% RSLogix 500 project TRAFFIC Multiple.RSS, saved by version 8.30.00.16 %
PROJECT "UNTITLED"    % processor: Bul.1763 MicroLogix 1100 Series B %

PROGRAM FILES
  LAD 2   8 rungs

DATA FILES
  O0 OUTPUT  4 elements
  I1 INPUT  6 elements
  S2 STATUS  66 elements
  B3 BINARY  1 elements
  T4 TIMER  7 elements
  C5 COUNTER  1 elements
  R6 CONTROL  1 elements
  N7 INTEGER  1 elements
  F8 FLOAT  1 elements

LADDER 2
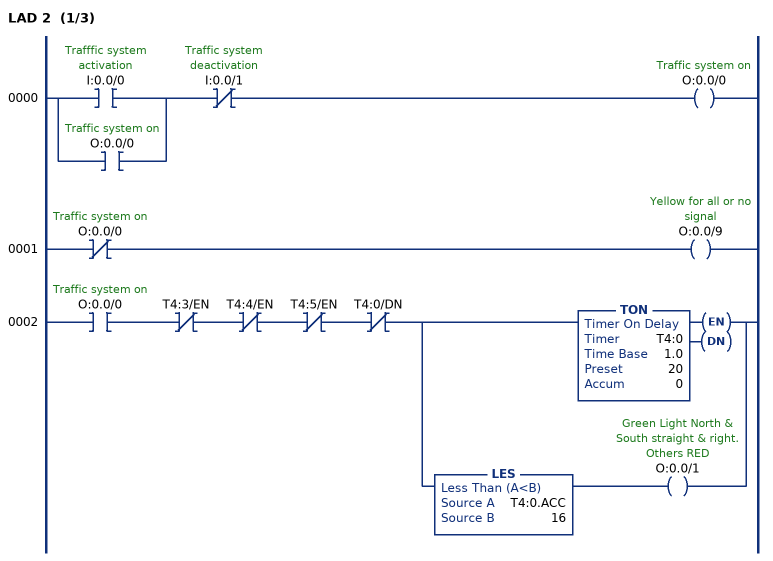
% Rung: 0 %
SOR BST XIC I:0.0/0 NXB XIC O:0.0/0 BND XIO I:0.0/1 OTE O:0.0/0 EOR
%   I:0.0/0  "Trafffic system activation" %
%   O:0.0/0  "Traffic system on" %
%   I:0.0/1  "Traffic system deactivation" %
% Rung: 1 %
SOR XIO O:0.0/0 OTE O:0.0/9 EOR
%   O:0.0/0  "Traffic system on" %
%   O:0.0/9  "Yellow for all or no signal" %
% Rung: 2 %
SOR XIC O:0.0/0 XIO T4:3/EN XIO T4:4/EN XIO T4:5/EN XIO T4:0/DN BST TON T4:0 1.0 20 0 NXB LES T4:0.ACC 16 OTE O:0.0/1 BND EOR
%   O:0.0/0  "Traffic system on" %
%   O:0.0/1  "Green Light North & South straight & right. Others RED" %

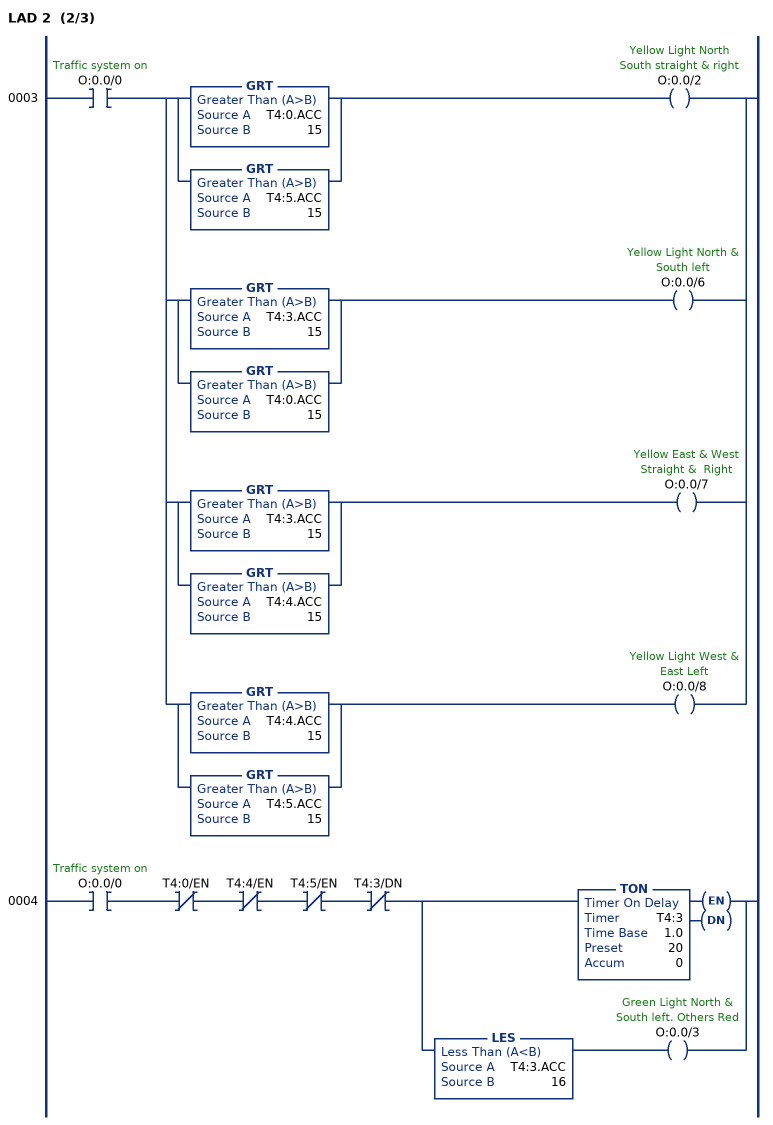
% Rung: 3 %
SOR XIC O:0.0/0 BST BST GRT T4:0.ACC 15 NXB GRT T4:5.ACC 15 BND OTE O:0.0/2 NXB BST BST GRT T4:3.ACC 15 NXB GRT T4:0.ACC 15 BND OTE O:0.0/6 NXB BST BST GRT T4:3.ACC 15 NXB GRT T4:4.ACC 15 BND OTE O:0.0/7 NXB BST GRT T4:4.ACC 15 NXB GRT T4:5.ACC 15 BND OTE O:0.0/8 BND BND BND EOR
%   O:0.0/0  "Traffic system on" %
%   O:0.0/2  "Yellow Light North South straight & right" %
%   O:0.0/6  "Yellow Light North & South left" %
%   O:0.0/7  "Yellow East & West Straight &  Right" %
%   O:0.0/8  "Yellow Light West & East Left" %
% Rung: 4 %
SOR XIC O:0.0/0 XIO T4:0/EN XIO T4:4/EN XIO T4:5/EN XIO T4:3/DN BST TON T4:3 1.0 20 0 NXB LES T4:3.ACC 16 OTE O:0.0/3 BND EOR
%   O:0.0/0  "Traffic system on" %
%   O:0.0/3  "Green Light North & South left. Others Red" %

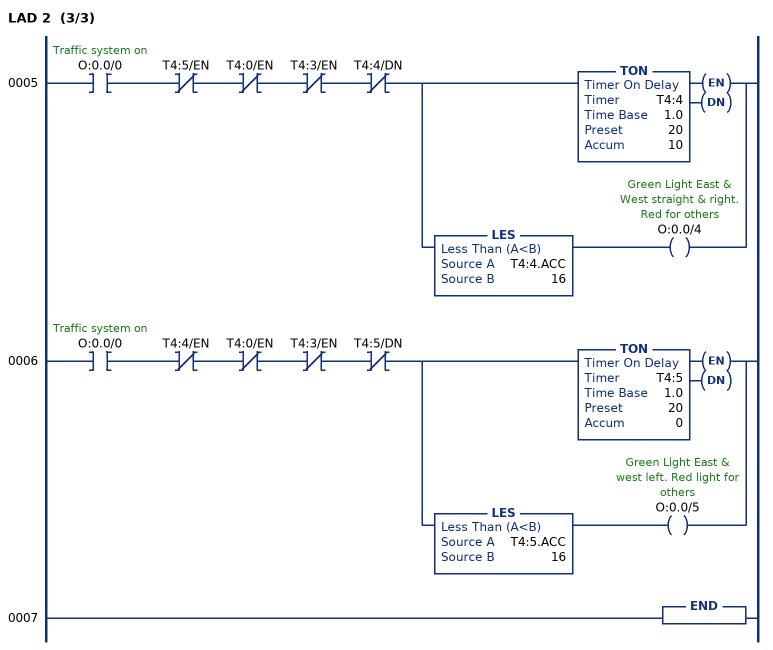
% Rung: 5 %
SOR XIC O:0.0/0 XIO T4:5/EN XIO T4:0/EN XIO T4:3/EN XIO T4:4/DN BST TON T4:4 1.0 20 10 NXB LES T4:4.ACC 16 OTE O:0.0/4 BND EOR
%   O:0.0/0  "Traffic system on" %
%   O:0.0/4  "Green Light East & West straight & right. Red for others" %
% Rung: 6 %
SOR XIC O:0.0/0 XIO T4:4/EN XIO T4:0/EN XIO T4:3/EN XIO T4:5/DN BST TON T4:5 1.0 20 0 NXB LES T4:5.ACC 16 OTE O:0.0/5 BND EOR
%   O:0.0/0  "Traffic system on" %
%   O:0.0/5  "Green Light East & west left. Red light for others" %
% Rung: 7 %
SOR END EOR

DATA TABLE (non-zero values as saved)
DATA T4
% .PRE .ACC %
% T4:0 % 20 0
% T4:1 % 10 10
% T4:2 % 3 0
% T4:3 % 20 0
% T4:4 % 20 10
% T4:5 % 20 0
% T4:6 % 5 5
